Yaskawa INFORM job: 3-PKT.JBI

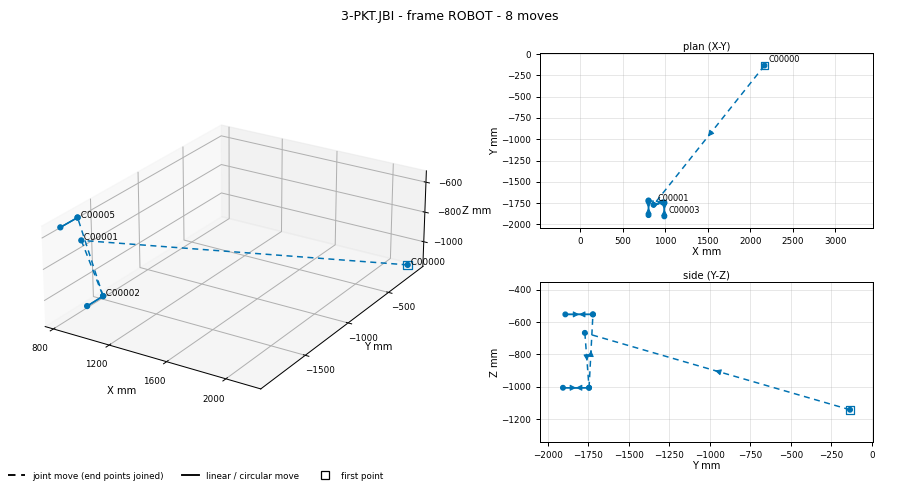
[picture p0: tool path of 3-PKT.JBI in frame ROBOT, 8 of 8 moves have a stored position in this frame; points joined in program order, loops and branches not executed]
/JOB
//NAME 3-PKT
//POS
///NPOS 8,8,8,0,0,0
///TOOL 0
///POSTYPE ROBOT
///RECTAN
///RCONF 0,0,0,0,1,0,0,0,0,0,0,0,0,0,0,0,0,0,0,0,0,0,0,0
C00000=2165.981,-134.012,-1141.311,-7.3017,-53.9175,4.0979
///RCONF 0,0,0,0,0,0,0,0,0,0,0,0,0,0,0,0,0,0,0,0,0,0,0,0
C00001=862.962,-1770.463,-666.772,-7.8640,-58.2964,-59.9433
C00002=989.763,-1744.422,-1005.573,-7.8743,-58.2989,-59.9312
C00003=989.740,-1905.474,-1005.598,-7.8696,-58.2984,-59.9363
C00004=989.763,-1744.422,-1005.573,-7.8743,-58.2989,-59.9312
C00005=804.137,-1720.593,-552.787,-7.8825,-58.2979,-59.9249
///RCONF 0,0,0,0,1,0,0,0,0,0,0,0,0,0,0,0,0,0,0,0,0,0,0,0
C00006=804.128,-1890.837,-552.801,-7.8828,-58.2979,-59.9247
///RCONF 0,0,0,0,0,0,0,0,0,0,0,0,0,0,0,0,0,0,0,0,0,0,0,0
C00007=804.137,-1720.593,-552.787,-7.8825,-58.2979,-59.9249
BC00000=385.118,3798.148,919.749
BC00001=385.118,3798.148,919.749
BC00002=385.118,3798.148,919.749
BC00003=385.118,3798.148,919.749
BC00004=385.118,3798.148,919.749
BC00005=385.118,3798.148,919.749
BC00006=385.118,3798.148,919.749
BC00007=385.118,3798.148,919.749
///POSTYPE PULSE
///PULSE
EC00000=2,1
EC00001=2,1
EC00002=2,1
EC00003=2,1
EC00004=2,1
EC00005=2,1
EC00006=2,1
EC00007=2,1
//INST
///DATE 2024/01/29 18:24
///ATTR SC,RW,RJ
////FRAME ROBOT
///GROUP1 RB1,BS1
///GROUP2 ST1
NOP
MOVJ C00000 BC00000 VJ=60.00  +MOVJ EC00000 VJ=90.00
MOVJ C00001 BC00001 VJ=90.00  +MOVJ EC00001 VJ=90.00
MOVJ C00002 BC00002 VJ=90.00  +MOVJ EC00002 VJ=90.00
MOVL C00003 BC00003 V=166.7  +MOVJ EC00003 VJ=90.00
MOVL C00004 BC00004 V=166.7  +MOVJ EC00004 VJ=90.00
MOVJ C00005 BC00005 VJ=90.00  +MOVJ EC00005 VJ=90.00
MOVL C00006 BC00006 V=166.7  +MOVJ EC00006 VJ=90.00
MOVL C00007 BC00007 V=166.7  +MOVJ EC00007 VJ=90.00
END
